(* CoDeSys 2.3 export: USER_PRG.EXP *)

(* POU SGL_Sismored/Sismored 4.0/New_telemetry_model/USER_PRG, FAI *)
PROGRAM USER_PRG
VAR
	xFirstCycle : BOOL := TRUE;
	aMaskLocalRemote : ARRAY [1..2] OF BOOL;
	eState : ARRAY [1..2] OF eStates;
	inst0Pack2LocalRemote : Pack2LocalRemote;
	inst0Check2LocalRemote : Check2LocalRemote;
	inst0Dev7SJ6x0 : Dev7SJ6x0;
	
END_VAR
(* body not read: x-want_COMMENT *)
END_PROGRAM
